// TIA Portal project "Speed Channels" (V18)

(* hardware
DEVICE "S7-1200 station_1"  S7-1200 Station
   slot 0: "Rack_0"  S7-1200 Rack  Rack  V1.0
   slot 1: "PLC_1"  CPU 1214C AC/DC/Rly  6ES7 214-1BG40-0XB0  V4.6
*)

// ===== PLC "PLC_1"  CPU 1214C AC/DC/Rly =====

VAR_GLOBAL   // PLC tag table "Default tag table"
   "Left_speed" AT %IW8 : Int;
   "Right_speed" AT %IW0 : Int;
   "GLL" AT %Q0.0 : Bool;
   "YLL" AT %Q0.1 : Bool;
   "RLL" AT %Q0.2 : Bool;
   "GLR" AT %Q0.3 : Bool;
   "YLR" AT %Q0.4 : Bool;
   "RLR" AT %Q0.5 : Bool;
END_VAR

FUNCTION "Block_2" : Void   // FC1, SCL
{ S7_Optimized_Access := 'TRUE' }
VERSION : 0.1
   VAR_INPUT
      LeftSpeedMemory : Int;
      RightSpeedMemory : Int;
   END_VAR
   VAR_OUTPUT
      GreenLightLeft : Bool;
      YellowLightLeft : Bool;
      RedLightLeft : Bool;
      GreenLightRight : Bool;
      YellowLightRight : Bool;
      RedLightRight : Bool;
   END_VAR
BEGIN
   // Check the speed for the left channel
   IF #LeftSpeedMemory > 80.0 THEN
       // Overspeeding: Activate red light
       #RedLightLeft := TRUE;
       #YellowLightLeft := FALSE;
       #GreenLightLeft := FALSE;
   ELSIF #LeftSpeedMemory >= 71.0 AND #LeftSpeedMemory <= 78.0 THEN
       // High speed warning: Activate yellow light
       #RedLightLeft := FALSE;
       #YellowLightLeft := TRUE;
       #GreenLightLeft := FALSE;
   ELSIF #LeftSpeedMemory < 70.0 AND #LeftSpeedMemory <> 0 THEN
       // Allowed speed: Activate green light
       #RedLightLeft := FALSE;
       #YellowLightLeft := FALSE;
       #GreenLightLeft := TRUE;

   ELSIF #LeftSpeedMemory = 0 THEN
       #RedLightLeft := FALSE;
       #YellowLightLeft := FALSE;
       #GreenLightLeft := FALSE;
   END_IF;

   // Check the speed for the right channel
   IF #RightSpeedMemory > 60.0 THEN
       // Overspeeding: Activate red light
       #RedLightRight := TRUE;
       #YellowLightRight := FALSE;
       #GreenLightRight := FALSE;
   ELSIF #RightSpeedMemory >= 50.0 AND #RightSpeedMemory <= 58.0 THEN
       // High speed warning: Activate yellow light
       #RedLightRight := FALSE;
       #YellowLightRight := TRUE;
       #GreenLightRight := FALSE;
   ELSIF #RightSpeedMemory < 49.0 AND #RightSpeedMemory <> 0 THEN
       // Allowed speed: Activate green light
       #RedLightRight := FALSE;
       #YellowLightRight := FALSE;
       #GreenLightRight := TRUE;
   ELSIF #RightSpeedMemory = 0 THEN
       #RedLightRight := FALSE;
       #YellowLightRight := FALSE;
       #GreenLightRight := FALSE;

   END_IF;
END_FUNCTION

ORGANIZATION_BLOCK "Main"   // OB1, LAD, ProgramCycle
TITLE = "Main Program Sweep (Cycle)"
{ S7_Optimized_Access := 'TRUE' }
VERSION : 0.1
   VAR_INPUT
      Initial_Call : Bool;   // Initial call of this OB
      Remanence : Bool;   // =True, if remanent data are available
   END_VAR
BEGIN

REGION Network 1
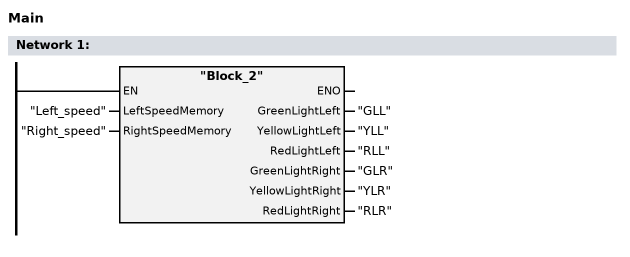
   RUNG wire#powerrail
      "Block_2"(LeftSpeedMemory := "Left_speed", RightSpeedMemory := "Right_speed", GreenLightLeft => "GLL", YellowLightLeft => "YLL", RedLightLeft => "RLL", GreenLightRight => "GLR", YellowLightRight => "YLR", RedLightRight => "RLR")
   END_RUNG
   // the same network as SCL:
   "Block_2"(LeftSpeedMemory := "Left_speed",
             RightSpeedMemory := "Right_speed",
             GreenLightLeft => "GLL",
             YellowLightLeft => "YLL",
             RedLightLeft => "RLL",
             GreenLightRight => "GLR",
             YellowLightRight => "YLR",
             RedLightRight => "RLR");
END_REGION
END_ORGANIZATION_BLOCK